FUNCTION_BLOCK App5_yAandyB (* Composite Function Block Type *)
  (* Standard: 61499-2 *)
  (* Version 0.0, 2018-11-06, 4DIAC-IDE, 4DIAC-Consortium *)
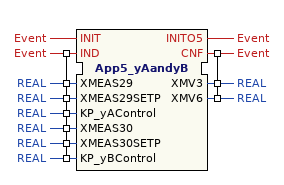
  EVENT_INPUT
    INIT; (* Initialization Request *)
    IND WITH XMEAS29, XMEAS29SETP, KP_yAControl, XMEAS30, XMEAS30SETP, KP_yBControl; (* Normal Execution Request *)
  END_EVENT
  EVENT_OUTPUT
    INITO5; (* Initialization Confirm *)
    CNF WITH XMV3, XMV6; (* Execution Confirmation *)
  END_EVENT
  VAR_INPUT
    XMEAS29 : REAL;
    XMEAS29SETP : REAL;
    KP_yAControl : REAL;
    XMEAS30 : REAL;
    XMEAS30SETP : REAL;
    KP_yBControl : REAL;
  END_VAR
  VAR_OUTPUT
    XMV3 : REAL;
    XMV6 : REAL;
  END_VAR
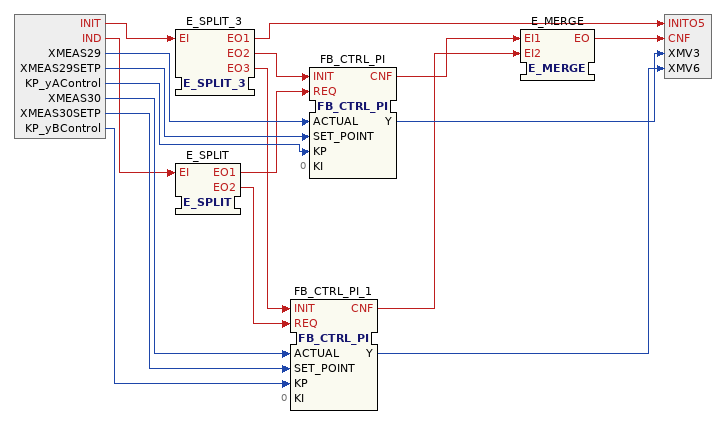
  FBS
    E_SPLIT_3 : E_SPLIT_3;
    E_SPLIT : E_SPLIT;
    FB_CTRL_PI : FB_CTRL_PI(KI := 0);
    FB_CTRL_PI_1 : FB_CTRL_PI(KI := 0);
    E_MERGE : E_MERGE;
  END_FBS
  EVENT_CONNECTIONS
    E_SPLIT_3.EO1 TO INITO5;
    E_SPLIT_3.EO2 TO FB_CTRL_PI.INIT;
    E_SPLIT_3.EO3 TO FB_CTRL_PI_1.INIT;
    E_SPLIT.EO1 TO FB_CTRL_PI.REQ;
    E_SPLIT.EO2 TO FB_CTRL_PI_1.REQ;
    FB_CTRL_PI.CNF TO E_MERGE.EI1;
    FB_CTRL_PI_1.CNF TO E_MERGE.EI2;
    E_MERGE.EO TO CNF;
    INIT TO E_SPLIT_3.EI;
    IND TO E_SPLIT.EI;
  END_CONNECTIONS
  DATA_CONNECTIONS
    FB_CTRL_PI.Y TO XMV3;
    FB_CTRL_PI_1.Y TO XMV6;
    XMEAS29 TO FB_CTRL_PI.ACTUAL;
    XMEAS29SETP TO FB_CTRL_PI.SET_POINT;
    KP_yAControl TO FB_CTRL_PI.KP;
    XMEAS30 TO FB_CTRL_PI_1.ACTUAL;
    XMEAS30SETP TO FB_CTRL_PI_1.SET_POINT;
    KP_yBControl TO FB_CTRL_PI_1.KP;
  END_CONNECTIONS
END_FUNCTION_BLOCK
